FUNCTION_BLOCK TcoExistsTask EXTENDS TcoDataTask
VAR
	_exists : BOOL;
END_VAR

SUPER^();

{attribute 'monitoring' := 'variable'}
PROPERTY Exists : BOOL
GET
Exists := _exists;
END_GET
END_PROPERTY

END_FUNCTION_BLOCK

(* stored: Version 1.1.0.1, ProductVersion 3.1.4024.9
   POU TcoExistsTask: Id {ec29d82c-42e7-05da-1463-9c768d234341}, SpecialFunc None
   Property Exists: Id {bb96b594-86d1-0ee3-3dec-35210736ed0b}
   Get Get: Id {376ffdd7-7453-0cd0-1692-fe1d9365ec51} *)
